TYPE ST_Event :
STRUCT
	Source:			I_Component;
	Instance:		STRING(255);
	Class:			STRING(255);
	EventType:		E_Event;
	Timestamp:   	ULINT;
	ID:				UDINT;
	Message:		STRING(255);
	Arguments:		STRING(255);
	Active:			BOOL;
	New:			BOOL;
END_STRUCT
END_TYPE

(* stored: Version 1.1.0.1
   DUT ST_Event: Id {424f55e5-b514-4649-8354-f5dfeb5cecd2} *)
